# EPICS autosave request: softGlueApp/Db/DivByN_settings.req
$(P)$(H)DivByN-$(N)_CLOCK_Signal
$(P)$(H)DivByN-$(N)_ENABLE_Signal
$(P)$(H)DivByN-$(N)_OUT_Signal
$(P)$(H)DivByN-$(N)_RESET_Signal
$(P)$(H)DivByN-$(N)_N
